INTERFACE ITF_BaseComponentDecoratorParent EXTENDS ITF_BaseComponent

END_INTERFACE

(* stored: Version 1.1.0.1, ProductVersion 3.1.4024.15
   Itf ITF_BaseComponentDecoratorParent: Id {ef036001-9570-432e-9bbf-6e35bc3c51a9} *)
